(* IEC 61131-3 sources: CodesysTest/alpha/export/FBs/Components/Load Plate/FB_BaseLoadPlate.pou/Internal/ExtendLoadPlate.prop, 1 file *)

(* ---- Get.pm.st ---- *)
(*#-#-#-#-#-#-#-#-#-#---Declaration---#-#-#-#-#-#-#-#-#-#-#-#-#*)

VAR
END_VAR
(*#-#-#-#-#-#-#-#-#-#---Implementation---#-#-#-#-#-#-#-#-#-#-#-#-#*)

ExtendLoadPlate := _manualOff OR ((_triggerActiveONS.OSF OR _shakeActiveONS.OSR OR _loadPlateInUseONS.OSR) AND inUse) OR ((_estopOK.OSR OR _disabledPositionHasUpdated OR _loadPlateInUseONS.OSF) AND disabledPosition = PackageEjectionDisabledPosition.LoadingPosition AND NOT inUse);
IF ExtendLoadPlate THEN
	RETURN;
END_IF
